// TIA Portal V19 export
DATA_BLOCK "MwFakCalc"   // DB133
// stored: InstanceOfName MwFakCalc_FB, InstanceOfType FB
"MwFakCalc_FB"
   // VAR_INPUT
   //    AreaInterface : "AreaInterface";
   //    ZSI : "udt_ZoneSafetyInterface";
   //    DSI : Struct
   //       PushAx : "udt_DeviceSafetyInterface";
   //       Gripper : "udt_DeviceSafetyInterface";
   //    END_STRUCT;
   //    Drive : Struct
   //       PushAx : "TAx_DriveInterface";
   //    END_STRUCT;
   //    HWID : Struct
   //       PushAx_TEL1 : HW_SUBMODULE;
   //    END_STRUCT;
   //    DataIn : Struct
   //       MaterialPresenceEntry : Bool;
   //       MaterialPresenceExit : Bool;
   //       MaterialJam : Bool;
   //       PushAx_Ls_HomeFwd : Bool;
   //       PushAx_Ls_RestBwd : Bool;
   //       PushAx_Ls_LowSpeedHome : Bool;
   //       PushAx_Ls_LowSpeedRest : Bool;
   //       PushAx_Ls_Touch : Bool;
   //       Gripper_Ls_ForceOpen : Bool;
   //       PushAx : "SpeedMachine_DataIn";
   //       Gripper : "ValveMachine_DataIn";
   //    END_STRUCT;
   //    CIn : Struct
   //       Manager : Struct
   //          EnableStopDoorOpeningReq : Bool;
   //          EnableStopInPhase : Bool;
   //          EnableStopProgrammed : Bool;
   //       END_STRUCT;
   //       Rollformer_Standstill : Bool;
   //       Rollformer_CheckNextFwd : Bool;
   //       Rollformer_CheckNextBwd : Bool;
   //       MW_ActualFAK : LReal;
   //       SemiAut_And_ButtonPressed : Bool;
   //       PostServo_MeasuredValueG : LReal;
   //       PostServo_MeasuredValueW : LReal;
   //       PostServo_MeasuredID : UInt;
   //    END_STRUCT;
   //    Config : Struct
   //       PushAx : "SpeedMachine_Config";
   //       Gripper : "ValveMachine_Config";
   //       MaterialPresenceDly : Time;
   //       MaterialAbsenceDly : Time;
   //       PushAx_FwdTimeout { ExternalAccessible := 'False'; ExternalVisible := 'False'; ExternalWritable := 'False'} : Time;
   //       PushAx_BwdTimeout { ExternalAccessible := 'False'; ExternalVisible := 'False'; ExternalWritable := 'False'} : Time;
   //       Default_FAK : LReal;
   //    END_STRUCT;
   // END_VAR
   // VAR_OUTPUT
   //    MachineInterface : "MachineInterface";
   //    DataOut : Struct
   //       PushAx : "SpeedMachine_DataOut";
   //       Gripper : "ValveMachine_DataOut";
   //       MeasInput_ExeReg : Bool;
   //    END_STRUCT;
   //    COut : Struct
   //       PushAx : "SpeedMachine_COut";
   //       Gripper : "ValveMachine_COut";
   //       StopMaterialFeeding : Bool;
   //       MW_FAK_ChangeIsRequest : Bool;
   //    END_STRUCT;
   // END_VAR
   // VAR_IN_OUT
   //    PersistentValues : "udt_MwFacCalc_Pers";
   //    TO_Gripper_Encoder : TO_ExternalEncoder;
   //    TO_Gripper_MeasInput : TO_MeasuringInput;
   //    TO_Wheel_MeasInput : TO_MeasuringInput;
   // END_VAR
   // VAR
   //    Sts : Struct
   //       PushAx : Struct
   //          LowSpeedRest : Bool;
   //          LowSpeedHome : Bool;
   //       END_STRUCT;
   //       Gripper : Struct
   //          OffsetPos : LReal;
   //          PosRel : LReal;
   //       END_STRUCT;
   //       AlarmPresence : Bool;
   //       Status : Int;
   //       MW_FAK_ChangeIsRequest : Bool;
   //       AverageFAKIsValid : Bool;
   //       WheelMeasInp_SaveIdLastPosEdge : UInt;
   //       GripperMeasInp_SaveIdLastPosEdge : UInt;
   //       GripperMeasInp_LastID : UInt;
   //       WheelMeasInp_LastID : UInt;
   //       PostServo_LastID : UInt;
   //    END_STRUCT;
   //    Ctrl : Struct
   //       StopInPhase : Bool;
   //       StopProgrammed : Bool;
   //       MeasuringStart : Bool;
   //       MeasInp_Enable : Bool;
   //       Meas1_Exe : Bool;
   //       Meas2_Exe : Bool;
   //       Gripper_RollformerForceOpen : Bool;
   //       Gripper_AutOpen : Bool;
   //       Gripper_AutClose : Bool;
   //       PushAx_AutFwd : Bool;
   //       PushAx_AutBwd : Bool;
   //       Rollformer_FwdEnable : Bool;
   //       Rollformer_BkwWnable : Bool;
   //       Rollformer_FastStop : Bool;
   //    END_STRUCT;
   //    Alarm : Struct
   //       PushAx_UnvalidStateLsZeroRest : Bool;
   //       PushAx_UnvalidStateLsLow : Bool;
   //       PushAx_LowSpeedHome_NotEngaged : Bool;
   //       PushAx_LowSpeedRest_NotEngaged : Bool;
   //       PushAx_TimeoutFwd : Bool;
   //       PushAx_TimeoutBwd : Bool;
   //       MaterialNoPresence : Bool;
   //       MaterialJamEntry : Bool;
   //       Meas1RegNotGet : Bool;
   //       Meas2RegNotGet : Bool;
   //       Gripper_MaxPosExceed : Bool;
   //       PushAx : "SpeedMachine_Alr";
   //       Gripper : "ValveAlr";
   //       Gripper_Encoder : "TExtEncoder_Alarms";
   //       Gripper_MeasInput : "TMeasuring_Alarms";
   //       Wheel_MeasInput : "TMeasuring_Alarms";
   //    END_STRUCT;
   //    Warning : Struct
   //       PushAx : "SpeedMachine_Wng";
   //       Gripper : "ValveMachine_Wng";
   //       MaterialNoPrresence : Bool;
   //    END_STRUCT;
   //    Diag : Struct
   //       Gripper_Encoder : "TO_Diagnostic";
   //       Gripper_MeasInput : "TO_Diagnostic";
   //       Wheel_MeasInput : "TO_Diagnostic";
   //    END_STRUCT;
   //    PushAx : "SpeedMachine_FB";
   //    Gripper : "ValveMachine_FB";
   //    Gripper_MeasInp { S7_SetPoint := 'True'} : "MeasuringInput";
   //    Wheel_MeasInp { S7_SetPoint := 'True'} : "MeasuringInput";
   //    MeasRegIEmpty { S7_SetPoint := 'True'} : "udt_MwFacCalc_RegItem";
   //    tonMaterialPresence : TON_TIME;
   //    tonMaterialAbsence : TON_TIME;
   //    tonPushAxFwd { S7_SetPoint := 'True'} : TON_TIME;
   //    tonPushAxBwd { S7_SetPoint := 'True'} : TON_TIME;
   //    tonRollformer_BwdCheckNext { S7_SetPoint := 'True'} : TON_TIME;
   // END_VAR
BEGIN
   AreaInterface.EStop := FALSE;
   AreaInterface.Man := TRUE;
   AreaInterface.Aut := FALSE;
   AreaInterface.Cycle := FALSE;
   AreaInterface.StopInPhase := FALSE;
   AreaInterface.StopProgrammed := FALSE;
   AreaInterface.RstAlarms := FALSE;
   AreaInterface.ManOneShot := FALSE;
   AreaInterface.AutOneShot := FALSE;
   AreaInterface.CycleOneShot := FALSE;
   AreaInterface.CheckAutReady := FALSE;
   MachineInterface.AutReady := FALSE;
   MachineInterface.Aborting := FALSE;
   MachineInterface.AckStopInPhase := FALSE;
   MachineInterface.AckStopProgrammed := FALSE;
   MachineInterface.MotionsStandStill := TRUE;
   MachineInterface.AlarmsPresence := FALSE;
   MachineInterface.WarningPresence := FALSE;
END_DATA_BLOCK
